//Res := Minuend - Subtrahend
FUNCTION Matrix_ElementDifference : BOOL
VAR_IN_OUT CONSTANT
	Minuend : Matrix;
	Subtrahend : Matrix;
END_VAR
VAR_IN_OUT
	Res : Matrix;
END_VAR
VAR
	I : UINT;
END_VAR

IF NOT(Minuend.IsEqualSize(Res)) OR Minuend.IsEmpty THEN
	Matrix_ElementDifference := FALSE;
	RETURN;
END_IF

IF NOT(Subtrahend.IsEqualSize(Res)) OR Subtrahend.IsEmpty THEN
	Matrix_ElementDifference := FALSE;
	RETURN;
END_IF

Matrix_ElementDifference := TRUE;

FOR I := 0 TO Res.Length - 1 DO
	Res.SetI(I,Minuend.GetI(I)-Subtrahend.GetI(I));
END_FOR

END_FUNCTION

(* stored: Version 1.1.0.1, ProductVersion 3.1.4024.9
   POU Matrix_ElementDifference: Id {f74edede-e315-0158-3390-9afe49ecc709}, SpecialFunc None *)
